Universal Robots PolyScope program: 03_Pick_Place_03_DIO_popup.urp

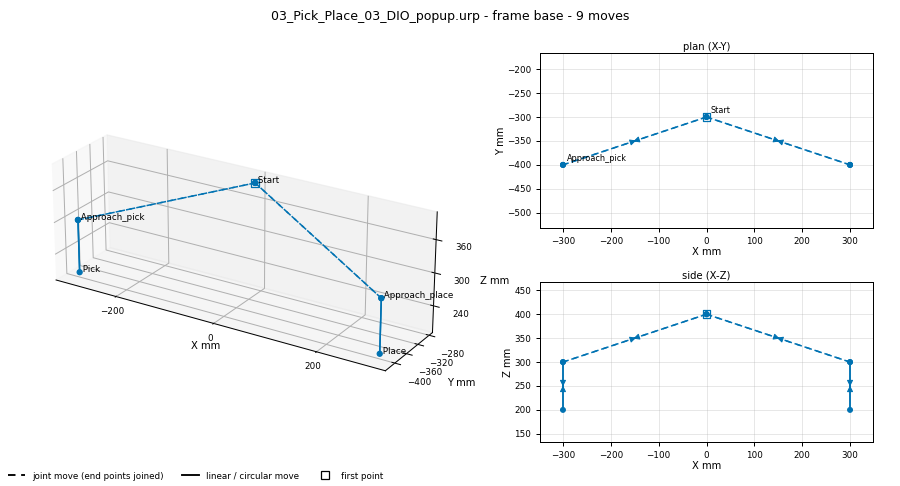
[picture p0: tool path of 03_Pick_Place_03_DIO_popup.urp in frame base, 9 of 9 moves have a stored position in this frame; points joined in program order, loops and branches not executed]
Program 03_Pick_Place_03_DIO_popup (installation=default directory=/home/ur/ursim-current/programs/Test_Programs createdIn=5.9.1.1031110 lastSavedIn=5.9.1.1031110 robotSerialNumber=20195599999)
Calibrated DH parameters: a=[0, -0.425, -0.3922, 0, 0, 0]; d=[0.1625, 0, 0, 0.1333, 0.0997, 0.0996]; alpha=[1.570796, 0, 0, 1.570796, -1.570796, 0]; deltaTheta=[0, 0, 0, 0, 0, 0]
Robot Program (runOnlyOnce=false)
  Wait DigitalInput pin=digital_in[0]; digitalValue=1
  MoveJ speed 60 deg/s, acceleration 80 deg/s^2 (useActiveTCP=true) feature=Base
    Waypoint Start: TCP in base x=0 y=-300 z=400 mm, rx=0 ry=3.1416 rz=0 rad; joints [-63.619, -58.456, -125.213, -86.33, 90, 26.381] deg
  Folder Pick
    MoveJ speed 60 deg/s, acceleration 80 deg/s^2 (useActiveTCP=true) feature=Base
      Waypoint Approach_pick: TCP in base x=-300 y=-400 z=300 mm, rx=0 ry=3.1416 rz=0 rad; joints [-111.408, -95.003, -113.354, -61.643, 90, -21.408] deg
    MoveL speed 250 mm/s, acceleration 1200 mm/s^2 (useActiveTCP=true) feature=Base
      Waypoint Pick: TCP in base x=-300 y=-400 z=200 mm, rx=0 ry=3.1416 rz=0 rad; joints [-111.408, -104.003, -120.574, -45.423, 90, -21.408] deg
      Set SingleDigitalPulseActionState SingleDigitalPulseActionState(hiPulseInSeconds=0.5, pin=digital_out[0])
      Waypoint Approach_pick: TCP in base x=-300 y=-400 z=300 mm, rx=0 ry=3.1416 rz=0 rad; joints [-111.408, -95.003, -113.354, -61.643, 90, -21.408] deg
    MoveJ speed 60 deg/s, acceleration 80 deg/s^2 (useActiveTCP=true) feature=Base
      Waypoint Start: TCP in base x=0 y=-300 z=400 mm, rx=0 ry=3.1416 rz=0 rad; joints [-63.619, -58.456, -125.213, -86.33, 90, 26.381] deg
  Folder Place
    MoveJ speed 60 deg/s, acceleration 80 deg/s^2 (useActiveTCP=true) feature=Base
      Waypoint Approach_place: TCP in base x=300 y=-400 z=300 mm, rx=0 ry=3.1416 rz=0 rad; joints [-37.668, -95.003, -113.354, -61.643, 90, 52.332] deg
    MoveL speed 250 mm/s, acceleration 1200 mm/s^2 (useActiveTCP=true) feature=Base
      Waypoint Place: TCP in base x=300 y=-400 z=200 mm, rx=0 ry=3.1416 rz=0 rad; joints [-37.668, -104.003, -120.574, -45.423, 90, 52.332] deg
      Set SingleDigitalPulseActionState SingleDigitalPulseActionState(hiPulseInSeconds=0.5, pin=digital_out[0])
      Waypoint Approach_place: TCP in base x=300 y=-400 z=300 mm, rx=0 ry=3.1416 rz=0 rad; joints [-37.668, -95.003, -113.354, -61.643, 90, 52.332] deg
    MoveJ speed 60 deg/s, acceleration 80 deg/s^2 (useActiveTCP=true) feature=Base
      Waypoint Start: TCP in base x=0 y=-300 z=400 mm, rx=0 ry=3.1416 rz=0 rad; joints [-63.619, -58.456, -125.213, -86.33, 90, 26.381] deg
  Folder Lamp
    Set DigitalOutput pin=digital_out[0]; digitalValue=1
    Wait Sleep waitTime=5
    Popup Message (haltProgram=false message=End Program inputType=Text)
